{attribute 'qualified_only'}
VAR_GLOBAL
	FluentString : fbFluentString;
END_VAR

(* stored: Version 1.1.0.1, ProductVersion 3.1.4024.2
   GVL Utils: Id {a5310a48-d7d0-4e88-b771-6ef37a06dbb7} *)
